{attribute 'strict'}
TYPE E_BufferInitState :
(
	BUFFER_INIT_ := 0
);
END_TYPE

(* stored: Version 1.1.0.1, ProductVersion 3.1.4024.9
   DUT E_BufferInitState: Id {29d363eb-8231-4512-acc9-715e702e3eeb} *)
